// Mitsubishi GX Works2 project: prpr1   PLC: Q03UDV

PROGRAM MAIN
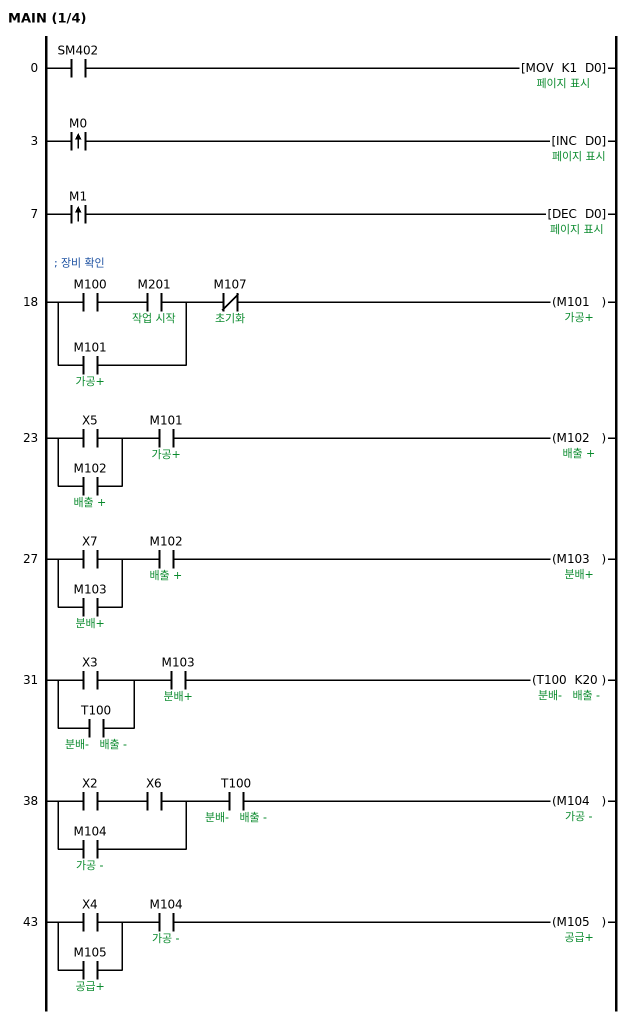
0     LD      SM402
      MOV     K1 D0  ; 페이지 표시
3     LDP     M0
      INC     D0
7     LDP     M1
      DEC     D0
; 장비 확인
18    LD      M100
      AND     M201  ; 작업 시작
      OR      M101  ; 가공+
      ANI     M107  ; 초기화
      OUT     M101  ; 가공+
23    LD      X5
      OR      M102  ; 배출 +
      AND     M101  ; 가공+
      OUT     M102  ; 배출 +
27    LD      X7
      OR      M103  ; 분배+
      AND     M102  ; 배출 +
      OUT     M103  ; 분배+
31    LD      X3
      OR      T100  ; 분배-   배출 -
      AND     M103  ; 분배+
      OUT     T100 K20  ; 분배-   배출 -
38    LD      X2
      AND     X6
      OR      M104  ; 가공 -
      AND     T100  ; 분배-   배출 -
      OUT     M104  ; 가공 -
43    LD      X4
      OR      M105  ; 공급+
      AND     M104  ; 가공 -
      OUT     M105  ; 공급+
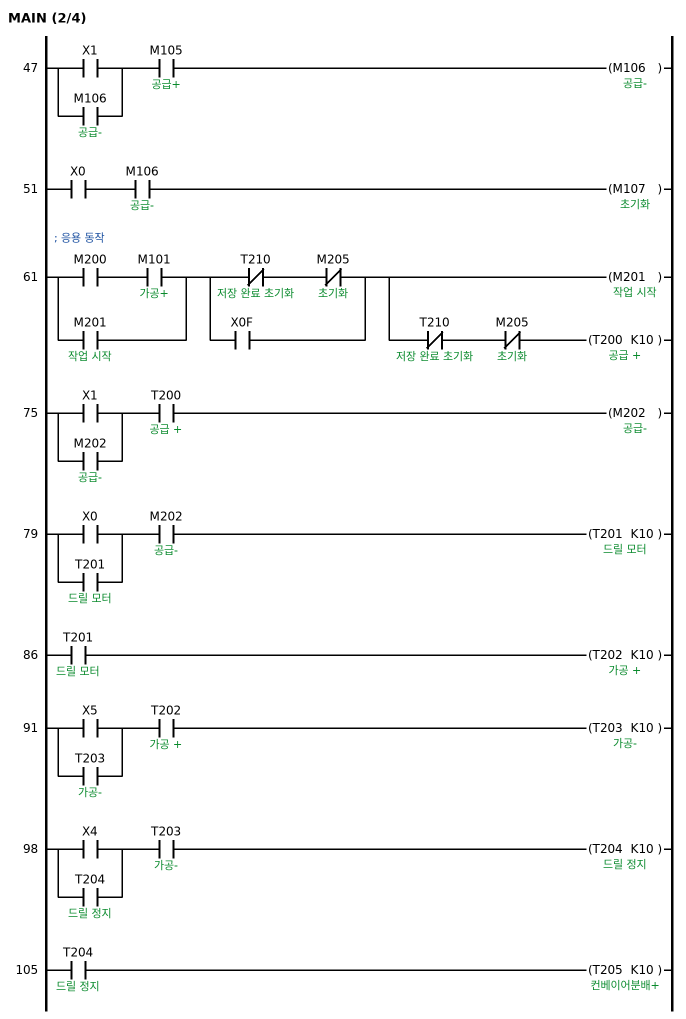
47    LD      X1
      OR      M106  ; 공급-
      AND     M105  ; 공급+
      OUT     M106  ; 공급-
51    LD      X0
      AND     M106  ; 공급-
      OUT     M107  ; 초기화
; 응용 동작
61    LD      M200
      AND     M101  ; 가공+
      OR      M201  ; 작업 시작
      LDI     T210  ; 저장 완료 초기화
      ANI     M205  ; 초기화
      OR      X0F
      ANB
      OUT     M201  ; 작업 시작
      ANI     T210  ; 저장 완료 초기화
      ANI     M205  ; 초기화
      OUT     T200 K10  ; 공급 +
75    LD      X1
      OR      M202  ; 공급-
      AND     T200  ; 공급 +
      OUT     M202  ; 공급-
79    LD      X0
      OR      T201  ; 드릴 모터
      AND     M202  ; 공급-
      OUT     T201 K10  ; 드릴 모터
86    LD      T201  ; 드릴 모터
      OUT     T202 K10  ; 가공 +
91    LD      X5
      OR      T203  ; 가공-
      AND     T202  ; 가공 +
      OUT     T203 K10  ; 가공-
98    LD      X4
      OR      T204  ; 드릴 정지
      AND     T203  ; 가공-
      OUT     T204 K10  ; 드릴 정지
105   LD      T204  ; 드릴 정지
      OUT     T205 K10  ; 컨베이어분배+
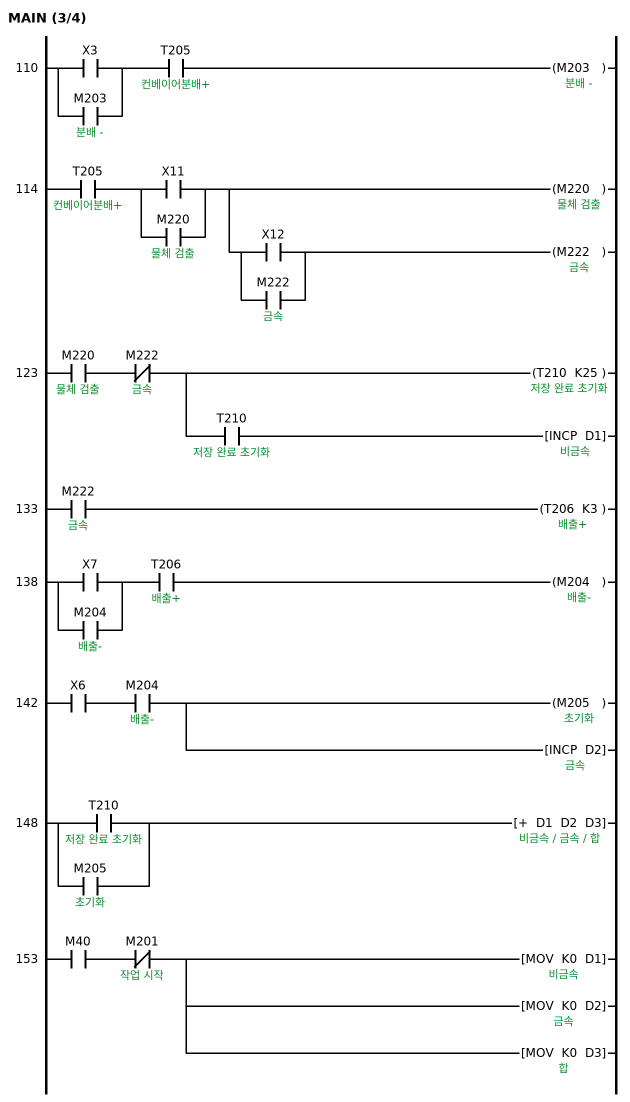
110   LD      X3
      OR      M203  ; 분배 -
      AND     T205  ; 컨베이어분배+
      OUT     M203  ; 분배 -
114   LD      T205  ; 컨베이어분배+
      LD      X11
      OR      M220  ; 물체 검출
      ANB
      OUT     M220  ; 물체 검출
      LD      X12
      OR      M222  ; 금속
      ANB
      OUT     M222  ; 금속
123   LD      M220  ; 물체 검출
      ANI     M222  ; 금속
      OUT     T210 K25  ; 저장 완료 초기화
      AND     T210  ; 저장 완료 초기화
      INCP    D1  ; 비금속
133   LD      M222  ; 금속
      OUT     T206 K3  ; 배출+
138   LD      X7
      OR      M204  ; 배출-
      AND     T206  ; 배출+
      OUT     M204  ; 배출-
142   LD      X6
      AND     M204  ; 배출-
      OUT     M205  ; 초기화
      INCP    D2  ; 금속
148   LD      T210  ; 저장 완료 초기화
      OR      M205  ; 초기화
      +       D1 D2 D3  ; 합
153   LD      M40
      ANI     M201  ; 작업 시작
      MOV     K0 D1
      MOV     K0 D2
      MOV     K0 D3
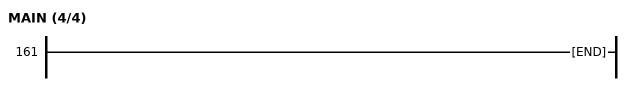
161   END
END_PROGRAM

PROGRAM OUTPUT
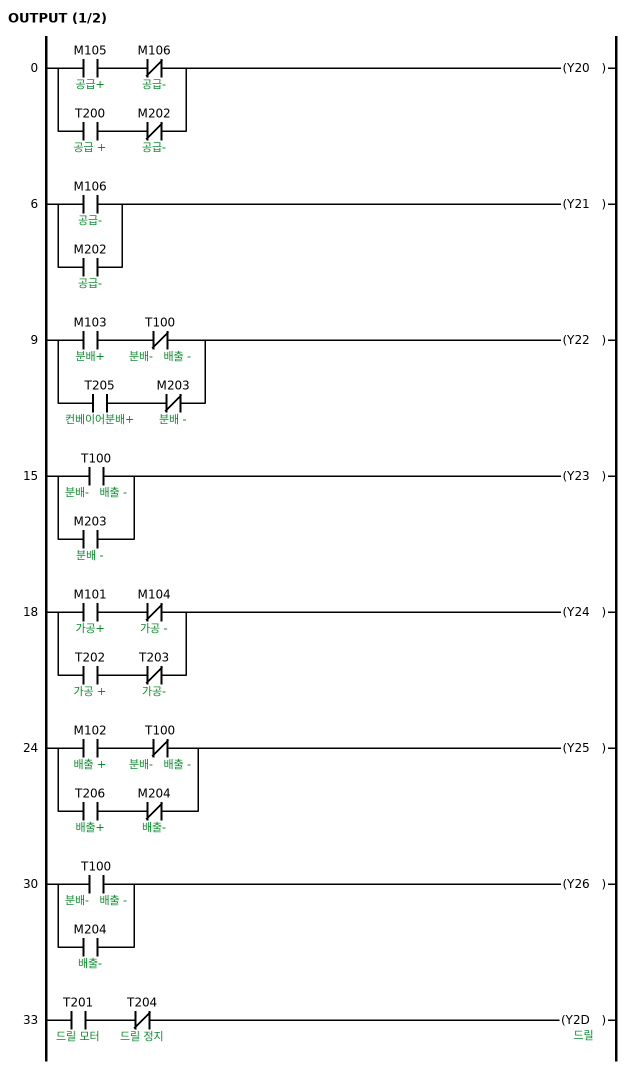
0     LD      M105  ; 공급+
      ANI     M106  ; 공급-
      LD      T200  ; 공급 +
      ANI     M202  ; 공급-
      ORB
      OUT     Y20
6     LD      M106  ; 공급-
      OR      M202  ; 공급-
      OUT     Y21
9     LD      M103  ; 분배+
      ANI     T100  ; 분배-   배출 -
      LD      T205  ; 컨베이어분배+
      ANI     M203  ; 분배 -
      ORB
      OUT     Y22
15    LD      T100  ; 분배-   배출 -
      OR      M203  ; 분배 -
      OUT     Y23
18    LD      M101  ; 가공+
      ANI     M104  ; 가공 -
      LD      T202  ; 가공 +
      ANI     T203  ; 가공-
      ORB
      OUT     Y24
24    LD      M102  ; 배출 +
      ANI     T100  ; 분배-   배출 -
      LD      T206  ; 배출+
      ANI     M204  ; 배출-
      ORB
      OUT     Y25
30    LD      T100  ; 분배-   배출 -
      OR      M204  ; 배출-
      OUT     Y26
33    LD      T201  ; 드릴 모터
      ANI     T204  ; 드릴 정지
      OUT     Y2D  ; 드릴
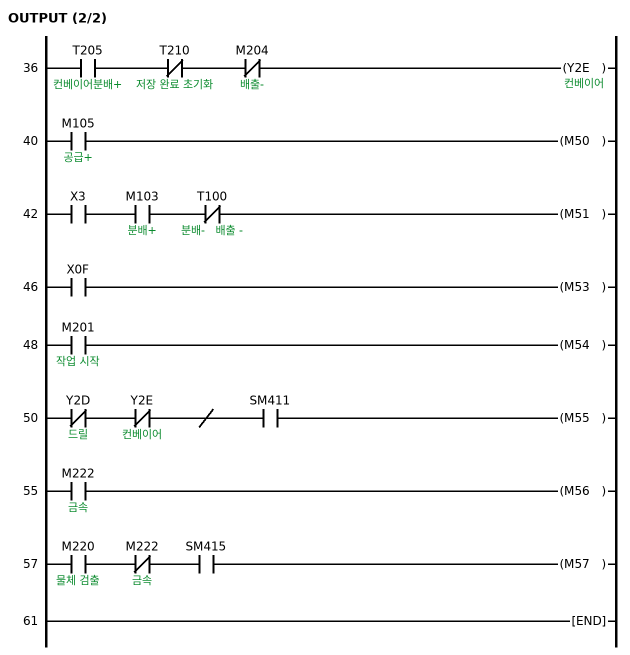
36    LD      T205  ; 컨베이어분배+
      ANI     T210  ; 저장 완료 초기화
      ANI     M204  ; 배출-
      OUT     Y2E  ; 컨베이어
40    LD      M105  ; 공급+
      OUT     M50
42    LD      X3
      AND     M103  ; 분배+
      ANI     T100  ; 분배-   배출 -
      OUT     M51
46    LD      X0F
      OUT     M53
48    LD      M201  ; 작업 시작
      OUT     M54
50    LDI     Y2D  ; 드릴
      ANI     Y2E  ; 컨베이어
      INV
      AND     SM411
      OUT     M55
55    LD      M222  ; 금속
      OUT     M56
57    LD      M220  ; 물체 검출
      ANI     M222  ; 금속
      AND     SM415
      OUT     M57
61    END
END_PROGRAM

// device comments not shown above
X15  ; 회전
X16  ; 회전 정지
X20  ; 가 모 버
X21  ; 컨 모 버
X22  ; 공 전 버
X30  ; 컨 모 버
X40  ; 공 전 버
X41  ; 공 후 버
Y0D  ; 드릴
M10  ; 공급 시작
M11  ; 공급 +
M12  ; 공급 -
M13  ; 초기화
M20  ; 가공 모드
M21  ; 가공 +
M22  ; 가공-
M30  ; 분배 작동
M31  ; 분배 +
M32  ; 분배-
T101  ; 배출 -
